FUNCTION_BLOCK FB_ClickLog
VAR
    startTimer : BOOL := FALSE;
    clickDetected : BOOL;
    elapsedTime : TIME;
    timer : TON;
    clickTimes : ARRAY[1..50] OF TIME;
    clickIndex : INT := 0;
    pauseTimer : TON;
	InputVariable AT %I* : BOOL;
END_VAR

// NIET GETEST - CHATGPT GEMAAKT

IF NOT startTimer THEN
    IF InputVariable THEN // Vervang 'InputVariable' door je daadwerkelijke input
        startTimer := TRUE;
        timer.IN := TRUE;
        timer.PT := T#5s;
        pauseTimer.PT := T#2s;
    END_IF;
ELSE
    timer();
    pauseTimer();

    IF timer.Q THEN
        pauseTimer.IN := TRUE;
        timer.IN := FALSE;
    ELSIF pauseTimer.Q THEN
        pauseTimer.IN := FALSE;
        timer.IN := TRUE;
    END_IF;

    IF InputVariable AND NOT pauseTimer.Q THEN
        IF clickIndex < 10 THEN
            clickIndex := clickIndex + 1;
            clickTimes[clickIndex] := timer.ET;
        END_IF;
    END_IF;
END_IF;

// Reset timer elapsed time at the start of each recording period
IF timer.IN THEN
    timer.IN := FALSE;
    timer(); // Update de timer status
    timer.IN := TRUE;
END_IF;

METHOD GetMinimumTime : TIME
VAR_INPUT
	    i : INT;
END_VAR

// NIET GETEST - CHATGPT GEMAAKT
// controleer in welke formaat time word gezet in de clicktimes array
GetMinimumTime := T#24D; // Stel een hoge beginwaarde in

FOR i := 1 TO clickIndex DO
	IF clickTimes[i] < GetMinimumTime THEN
		GetMinimumTime := clickTimes[i];
	END_IF;
END_FOR;
END_METHOD

END_FUNCTION_BLOCK

(* stored: Version 1.1.0.1, ProductVersion 3.1.4024.12
   POU FB_ClickLog: Id {8f6cddd7-835e-492b-b772-11d3f86c5c82}, SpecialFunc None
   Method GetMinimumTime: Id {0ac996dc-da40-4a57-831c-438a84555969} *)
